// TIA Portal V17 export
// export: Created 2024-06-14T09:53:49.5467577Z, ExportSetting WithDefaults, DisplayName Totally Integrated Automation Portal, DisplayVersion V17, DisplayName TIA Portal Openness, DisplayVersion V17, DisplayName TIA Portal Version Control Interface, DisplayVersion V17, DisplayName Simotion SCOUT TIA, DisplayVersion 5.4.3.0, DisplayName SINAMICS Startdrive Advanced, DisplayVersion V17 SP1 Update 1, DisplayName SINAMICS Startdrive G110M, G120, G120C, G120D, G120P, G115D, DisplayVersion V17 SP1 Update 1, DisplayName SINAMICS Startdrive G130, G150, S120, S150, SINAMICS MV, S210, DisplayVersion V17 SP1 Update 1, DisplayName STEP 7 Professional, DisplayVersion V17, DisplayName STEP 7 Safety, DisplayVersion V17, DisplayName WinCC Professional, DisplayVersion V17
VAR_GLOBAL   // PLC tag table "Check Scale Station-6"
   TAG_201 AT %M2.3 : Bool;
   TAG_202 AT %M2.4 : Bool;
   Tag_100 AT %M2.5 : Bool;
   "anti jammer_L2" AT %M2.6 : Bool;
   Tag_79_L2 AT %M2.7 : Bool;
   S5_STOPPER_SENSOR_l2 AT %M3.0 : Bool;
   S5_SENSOR_CYL7_DUMMY_TAG AT %M3.1 : Bool;
   Tag_102 AT %M3.2 : Bool;
   Seq_Lifttable_done_L2 AT %M3.3 : Bool;
   MC_Reset_L2 AT %M3.4 : Bool;
   TAG_203 AT %M3.5 : Bool;
   TAG_204 AT %M3.6 : Bool;
   TAG_205 AT %M3.7 : Bool;
   TAG_206 AT %M4.0 : Bool;
   TAG_207 AT %M4.1 : Bool;
   TAG_208 AT %M4.2 : Bool;
   TAG_209 AT %M4.3 : Bool;
   TAG210 AT %M4.4 : Bool;
   TAG211 AT %M4.5 : Bool;
   TAG216 AT %M4.6 : Bool;
   TAG213 AT %M4.7 : Bool;
   TAG214 AT %M5.0 : Bool;
   TAG215 AT %M5.1 : Bool;
   TAG217 AT %M5.2 : Bool;
   TAG218 AT %M5.3 : Bool;
   TAG212 AT %M5.4 : Bool;
   old_id AT %MW6 : Int;
   New_id AT %MW18 : Int;
END_VAR
